// TIA Portal V18 export
// export: Created 2026-06-09T02:47:52.5453343Z, ExportSetting WithDefaults, DisplayName Totally Integrated Automation Portal, DisplayVersion V18, DisplayName TIA Portal Openness, DisplayVersion V18, DisplayName TIA Portal Version Control Interface, DisplayVersion V18, DisplayName STEP 7 Professional, DisplayVersion V18, DisplayName STEP 7 Safety, DisplayVersion V18, DisplayName WinCC Professional, DisplayVersion V18
VAR_GLOBAL   // PLC tag table "Zakrecarka"
   start_zakrecarka AT %M101.0 : Bool;
   stop_zakrecarka AT %M101.1 : Bool;
   cz_pojemnosciowy_zak AT %M201.0 : Bool;
   tasma_zakrecarka AT %Q0.4 : Bool;
   zakretka AT %Q0.3 : Bool;
   lampa_sygnalizacyjna AT %Q0.5 : Bool;
END_VAR
